(* PLC project Generated.project, CODESYS CODESYS V3.5 SP19 Patch 1 *)
(* stored: creationDateTime 2026-08-30T22:32:01.335763, modificationDateTime 2026-08-30T22:32:01.335763 *)

(* ======================================================================= ST_fbDiveSearch_Config - Reglages du cycle de recherche du fond ======================================================================= *)
TYPE ST_fbDiveSearch_Config : STRUCT
  DiveSpeedMin_Mps : REAL := 0.15;  (* Vitesse minimale de calcul du timeout (m/s) *)
  TimeoutMarginFactor : REAL := 1.5;  (* Marge appliquee au temps theorique *)
  TimeoutMinCourse_M : REAL := 1;  (* Course minimale prise en compte (m) *)
  TimeoutMaxCourse_M : REAL := 200;  (* Course maximale prise en compte (m) *)
  SecToMs : REAL := 1000;  (* Conversion secondes vers millisecondes *)
END_STRUCT;
END_TYPE
